FUNCTION_BLOCK FB_GenericLogger EXTENDS FB_GenericObserver IMPLEMENTS I_Logger		// Logger where real implementations can subscribe too
																					// This logger by itself does nothing
VAR
	// These VARs cannot be locally inside the METHODs since Twincat does not like that (will crash)
	helperPtr:					POINTER TO BYTE;	// Helper pointer to get the address of the interface
	helperIf:					I_Logger;	// Helper interface for casting back from POINTER TO BOOL to this interface
END_VAR
VAR PERSISTENT
	initCalled: 	INT;
	reInitCalled:	INT;
	exitCalled:		INT;
END_VAR

METHOD PUBLIC debug : BOOL	// Logs the data with log level 'DEBUG'
VAR_INPUT
	iData:		T_DEFAULT_STR;						// Data to be logged, limited to 255 characters
END_VAR
VAR
	i:				INT;
END_VAR
getObservers();
FOR i := 0 TO validObservers.cnt -1 BY 1 DO
	MEMCPY(ADR(helperIf), ADR(validObservers.observers[i].observer), 16);
	helperIf.debug(iData);
END_FOR
END_METHOD

METHOD PUBLIC deregister : BOOL
VAR_INPUT
	iWho:				T_SHORT_STR;
END_VAR
deregisterObserver(iWho);
END_METHOD

METHOD PUBLIC doLog : BOOL	// Logs the data with log level 'WARN'
VAR_INPUT
	iData:		T_DEFAULT_STR;						// Data to be logged, limited to 255 characters
	iLevel:		E_LOG_LEVEL := E_LOG_LEVEL.ERROR;	// Log level
END_VAR
VAR
	i:				INT;
END_VAR
getObservers();
FOR i := 0 TO validObservers.cnt -1 BY 1 DO
	MEMCPY(ADR(helperIf), ADR(validObservers.observers[i].observer), 16);
	helperIf.doLog(iData, iLevel);
END_FOR
END_METHOD

METHOD PUBLIC error : BOOL	// Logs the data with log level 'ERROR'
VAR_INPUT
	iData:		T_DEFAULT_STR;						// Data to be logged, limited to 255 characters
END_VAR
VAR
	i:				INT;
END_VAR
getObservers();
FOR i := 0 TO validObservers.cnt -1 BY 1 DO
	MEMCPY(ADR(helperIf), ADR(validObservers.observers[i].observer), 16);
	helperIf.error(iData);
END_FOR
END_METHOD

METHOD FB_exit : BOOL
VAR_INPUT
	bInCopyCode : BOOL; // if TRUE, the exit method is called for exiting an instance that is copied afterwards (online change).
END_VAR
IncInt(exitCalled);
END_METHOD

METHOD FB_init : BOOL
VAR_INPUT
	bInitRetains : BOOL; // if TRUE, the retain variables are initialized (warm start / cold start)
	bInCopyCode : BOOL;  // if TRUE, the instance afterwards gets moved into the copy code (online change)
END_VAR
IncInt(initCalled);
END_METHOD

METHOD FB_reinit : BOOL
IncInt(reInitCalled);
END_METHOD

METHOD PUBLIC info : BOOL	// Logs the data with log level 'INFO'
VAR_INPUT
	iData:		T_DEFAULT_STR;						// Data to be logged, limited to 255 characters
END_VAR
VAR
	i:				INT;
END_VAR
getObservers();
FOR i := 0 TO validObservers.cnt -1 BY 1 DO
	MEMCPY(ADR(helperIf), ADR(validObservers.observers[i].observer), 16);
	helperIf.info(iData);
END_FOR
END_METHOD

METHOD PUBLIC register : BOOL
VAR_INPUT
	iWho:		T_SHORT_STR;
	iObserver:	I_Logger;
END_VAR
VAR
	pointerSize:	UINT;
END_VAR
// Get the pointer value from the observer Interface

pointerSize := SIZEOF(helperPtr);
MEMCPY(ADR(helperPtr), ADR(iObserver), pointerSize);

registerObserver(iWho, helperPtr);
END_METHOD

METHOD PUBLIC trace : BOOL	// Logs the data with log level 'TRACE'
VAR_INPUT
	iData:		T_DEFAULT_STR;						// Data to be logged, limited to 255 characters
END_VAR
VAR
	i:				INT;
END_VAR
getObservers();
FOR i := 0 TO validObservers.cnt -1 BY 1 DO
	MEMCPY(ADR(helperIf), ADR(validObservers.observers[i].observer), 16);
	helperIf.trace(iData);
END_FOR
END_METHOD

METHOD PUBLIC warn : BOOL	// Logs the data with log level 'WARN'
VAR_INPUT
	iData:		T_DEFAULT_STR;						// Data to be logged, limited to 255 characters
END_VAR
VAR
	i:				INT;
END_VAR
getObservers();
FOR i := 0 TO validObservers.cnt -1 BY 1 DO
	MEMCPY(ADR(helperIf), ADR(validObservers.observers[i].observer), 16);
	helperIf.warn(iData);
END_FOR
END_METHOD

END_FUNCTION_BLOCK

(* stored: Version 1.1.0.1, ProductVersion 3.1.4026.18
   POU FB_GenericLogger: Id {6b7afa9a-3ef0-4064-9aa6-df93e70cdadd}, SpecialFunc None
   Method debug: Id {8c2b2095-4d21-428f-a8e3-a18f878ff344}
   Method deregister: Id {12e6bb0c-b52c-41f8-9013-d668763275b8}
   Method doLog: Id {76917e7c-d997-414e-a2cc-1bbec756b113}
   Method error: Id {9372b437-fd20-4858-a1e7-3c5de82cdadb}
   Method FB_exit: Id {fabba264-0aec-4c1f-9efa-4ea5f945b072}
   Method FB_init: Id {0f959e5c-f8e8-4694-a02f-8883e4af8964}
   Method FB_reinit: Id {1d1c27b1-2f56-44ca-a823-44c8362c8104}
   Method info: Id {1827ca1c-1baf-45da-a80a-61f73a6cfda8}
   Method register: Id {9f7a42cd-fcad-4024-ab3b-8224601a2510}
   Method trace: Id {613cae8c-5b42-4c04-afb9-cea7ddde6b2b}
   Method warn: Id {0a544c5c-2701-4121-abe0-731ebcbf45fa} *)
